TYPE "JB_Manager"
VERSION : 0.1
// Block: JB_Manager
   STRUCT
      Torch : Positioning_DOL_Machine_Manager;
      ClampEntry : ValveMachine_Manager;
      ClampExit : ValveMachine_Manager;
      CutHead : ValveMachine_Manager;
      PinchRoll_Feed : SpeedMachine_CIn_Manager;
      Pinchroll_Lift : ValveMachine_Manager;
      WeldingSetUp : JB_WeldingSetUp;
      ExtraLowON : Bool;
      ExtraLowPercentage : Real;
   END_STRUCT;

END_TYPE
